SUBAPPLICATION Uebung_039 (* Spiegelabfolge V2 mit Schrittkette *)
  (* Standard: 61499-2; Description: Copyright (c) 2023 Meisterschulen am Ostbahnhof This program and the accompanying materials are made available under the terms of the Eclipse Public License 2.0 which is available at https://www.eclipse.org/legal/epl-2.0/ SPDX-License-Identifier: EPL-2.0 Spiegelabfolge V2 mit Schrittkette geeignet für hydraulische 4/3 Wege Ventile oder pneumatische 5/3 Wege Ventile jeweils Mittelstellung gesperrt. *)
  (* Version 1.0, 2023-10-23, Franz Höpfinger, Meisterschulen am Ostbahnhof *)
  IMPORT logiBUS::io::DI::logiBUS_DI;
  IMPORT logiBUS::io::DQ::logiBUS_DO;
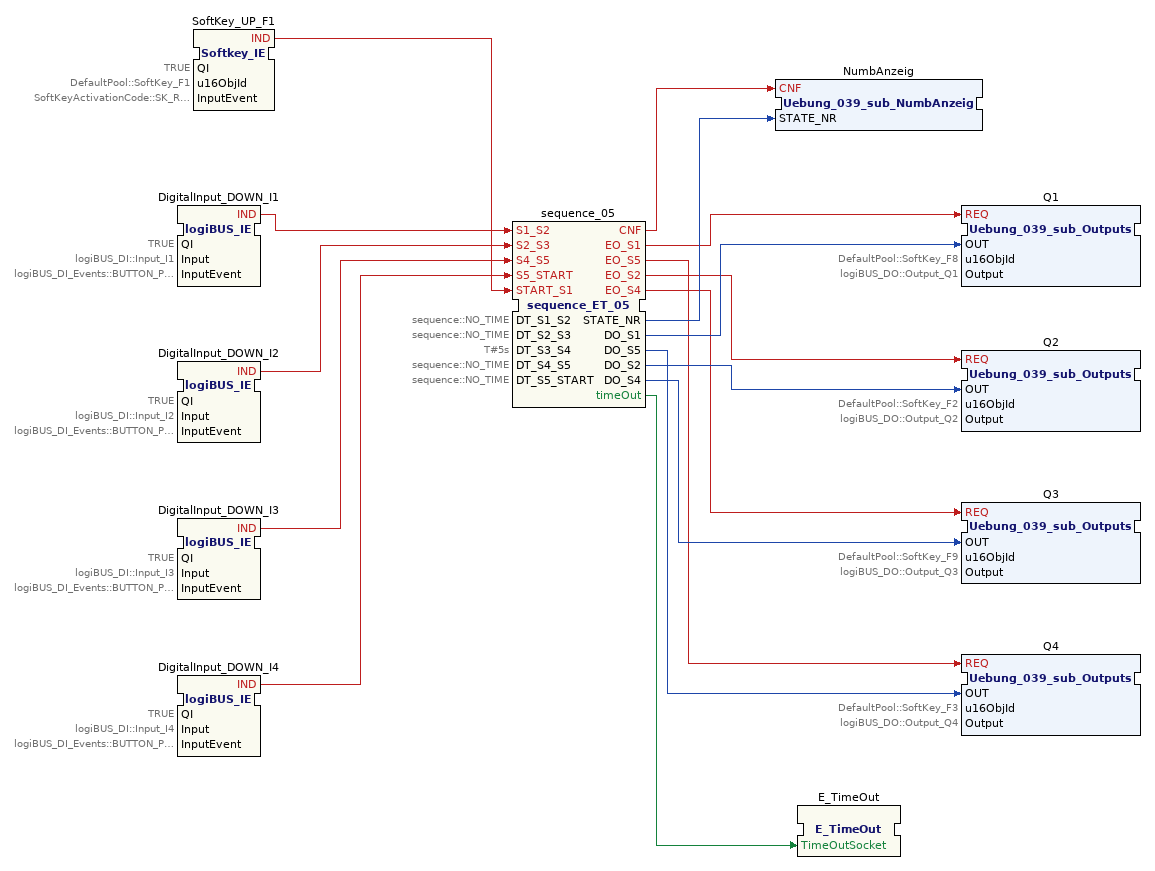
  FBS
    E_TimeOut : iec61499::events::E_TimeOut;
    DigitalInput_DOWN_I1 : logiBUS::io::DI::logiBUS_IE(QI := TRUE, Input := logiBUS_DI::Input_I1, InputEvent := logiBUS_DI_Events::BUTTON_PRESS_DOWN);
    DigitalInput_DOWN_I2 : logiBUS::io::DI::logiBUS_IE(QI := TRUE, Input := logiBUS_DI::Input_I2, InputEvent := logiBUS_DI_Events::BUTTON_PRESS_DOWN);
    DigitalInput_DOWN_I3 : logiBUS::io::DI::logiBUS_IE(QI := TRUE, Input := logiBUS_DI::Input_I3, InputEvent := logiBUS_DI_Events::BUTTON_PRESS_DOWN);
    DigitalInput_DOWN_I4 : logiBUS::io::DI::logiBUS_IE(QI := TRUE, Input := logiBUS_DI::Input_I4, InputEvent := logiBUS_DI_Events::BUTTON_PRESS_DOWN);
    sequence_05 : sequence_ET_05(DT_S1_S2 := sequence::NO_TIME, DT_S2_S3 := sequence::NO_TIME, DT_S3_S4 := T#5s, DT_S4_S5 := sequence::NO_TIME, DT_S5_START := sequence::NO_TIME);
    SoftKey_UP_F1 : Softkey_IE(QI := TRUE, u16ObjId := DefaultPool::SoftKey_F1, InputEvent := SoftKeyActivationCode::SK_RELEASED);
  END_FBS
  SUBAPPS
    NumbAnzeig : Uebung_039_sub_NumbAnzeig;
    Q1 : Uebung_039_sub_Outputs(u16ObjId := DefaultPool::SoftKey_F8, Output := logiBUS_DO::Output_Q1);
    Q4 : Uebung_039_sub_Outputs(u16ObjId := DefaultPool::SoftKey_F3, Output := logiBUS_DO::Output_Q4);
    Q2 : Uebung_039_sub_Outputs(u16ObjId := DefaultPool::SoftKey_F2, Output := logiBUS_DO::Output_Q2);
    Q3 : Uebung_039_sub_Outputs(u16ObjId := DefaultPool::SoftKey_F9, Output := logiBUS_DO::Output_Q3);
  END_SUBAPPS
  EVENT_CONNECTIONS
    DigitalInput_DOWN_I1.IND TO sequence_05.S1_S2;
    DigitalInput_DOWN_I2.IND TO sequence_05.S2_S3;
    DigitalInput_DOWN_I3.IND TO sequence_05.S4_S5;
    DigitalInput_DOWN_I4.IND TO sequence_05.S5_START;
    sequence_05.CNF TO NumbAnzeig.CNF;
    SoftKey_UP_F1.IND TO sequence_05.START_S1;
    sequence_05.EO_S1 TO Q1.REQ;
    sequence_05.EO_S5 TO Q4.REQ;
    sequence_05.EO_S2 TO Q2.REQ;
    sequence_05.EO_S4 TO Q3.REQ;
  END_CONNECTIONS
  DATA_CONNECTIONS
    sequence_05.STATE_NR TO NumbAnzeig.STATE_NR;
    sequence_05.DO_S1 TO Q1.OUT;
    sequence_05.DO_S5 TO Q4.OUT;
    sequence_05.DO_S2 TO Q2.OUT;
    sequence_05.DO_S4 TO Q3.OUT;
  END_CONNECTIONS
  ADAPTER_CONNECTIONS
    sequence_05.timeOut TO E_TimeOut.TimeOutSocket;
  END_CONNECTIONS
END_SUBAPPLICATION
